FUNCTION_BLOCK FB_GenericBrand_Transceiver EXTENDS FB_PressureSensor
VAR_INPUT
END_VAR
VAR_OUTPUT
END_VAR
VAR
END_VAR

METHOD getSignal : LREAL
VAR_INPUT
END_VAR
// Pressure Transducer
 // Using 4..20mA input card with a 0-10v sensor. To make this possible a 500ohm resister was added. Best to buy the correct hardware.
 // Scale 4.20mA value to 2v-10v
fBufferedSignal := Scale(signal := fInputSignal,
                           inputMin := 0.0, // 4mA
                           inputMax := 32767.0, // 20mA
                           outputMin := 2, // 2v at 4mA
                           outputMax := 10);

getSignal := fBufferedSignal;
END_METHOD

METHOD setSignal : BOOL
VAR_INPUT
    input : LREAL;
END_VAR
fInputSignal := input;
END_METHOD

END_FUNCTION_BLOCK

(* stored: Version 1.1.0.1, ProductVersion 3.1.4024.9
   POU FB_GenericBrand_Transceiver: Id {cd4b1846-ce79-448b-abe8-a8fbe7c0c982}, SpecialFunc None
   Method getSignal: Id {f6943603-3525-457e-9cd6-f74e6ed8300a}
   Method setSignal: Id {36be2125-0b4a-48c6-b8bd-0097dac38cec} *)
